FUNCTION_BLOCK SYMLINKMULTIVARDST_5A03F112CD5D470 (* Multiple variables single value symbolic link destination FB *)
  (* Standard: 61499-2 *)
  (* Version 1.0, 2008-10-02, milos, nxtControl GmbH, template *)
  PACKAGE Main;
  (* Compiler Cpp *)
  {SET_ATTRIBUTE(Runtime.FBType.ImplementingType, Runtime.System#DYNGEN_SYMLINKMVAR)}
  {SET_ATTRIBUTE(Configuration.GenericFBType.InterfaceParams, Runtime.System#I:=1;VALUE${I$}:INT)}
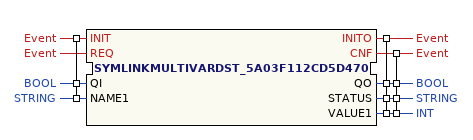
  EVENT_INPUT
    INIT WITH QI, NAME1; (* Initializes the symbolic link data destination FB with N (1 <= N <= 16) variables *)
    REQ; (* Explicit data read request *)
  END_EVENT
  EVENT_OUTPUT
    INITO WITH QO, STATUS, VALUE1; (* Initialization confirm *)
    CNF WITH QO, STATUS, VALUE1; (* Confirmation of an explicit or implicit data read request *)
  END_EVENT
  VAR_INPUT
    QI : BOOL; (* INIT event input qualifier *)
    NAME1 : STRING := '$${PATH}'; (* Names a symbolic link variable *)
  END_VAR
  VAR_OUTPUT
    QO : BOOL; (* Output event qualifier *)
    STATUS : STRING; (* FB status indicator *)
    VALUE1 : INT; (* Current value(i) in the named variable array element *)
  END_VAR
  EC_STATES
    START;
  END_STATES
END_FUNCTION_BLOCK
